// Mitsubishi GX Works2 project: SmartFarmDXST   PLC: FX3U/FX3UC

// global labels: Global1
VAR_GLOBAL
  v1 enb AT M130 : BOOL;
  v1 mode slc AT M131 : BOOL;
  v1 man OD AT M132 : BOOL;
  v1 Temp1 AT M133 : BOOL;
  v1 Temp2 AT M134 : BOOL;
  v1 Humid1 AT M135 : BOOL;
  v1 Humid2 AT M136 : BOOL;
  v1 Time1 AT M137 : BOOL;
  v1 Time2 AT M138 : BOOL;
  v1 Time3 AT M139 : BOOL;
  v1 Time4 AT M140 : BOOL;
  v1 AMB config AT M141 : BOOL;
  v1 TIME config AT M142 : BOOL;
  v1 con pass flg AT M144 : BOOL;
  v1 Drv flg AT M145 : BOOL;
  v1 Yman OD AT M146 : BOOL;
  v1 run dur AT D102 : INT;
  v1 rest dur AT D103 : INT;
  v0 enb AT M100 : BOOL;
  v0 mode slc AT M101 : BOOL;
  v0 man OD AT M102 : BOOL;
  v0 Temp1 AT M103 : BOOL;
  v0 Temp2 AT M104 : BOOL;
  v0 Humid1 AT M105 : BOOL;
  v0 Humid2 AT M106 : BOOL;
  v0 Time1 AT M107 : BOOL;
  v0 Time2 AT M108 : BOOL;
  v0 Time3 AT M109 : BOOL;
  v0 Time4 AT M110 : BOOL;
  v0 AMB config AT M111 : BOOL;
  v0 TIME config AT M112 : BOOL;
  v0 con kill flg AT M113 : BOOL;
  v0 con pass flg AT M114 : BOOL;
  v0 Drv flg AT M115 : BOOL;
  v0 run dur AT D100 : INT;
  v0 rest dur AT D101 : INT;
  v0 Yman OD AT M116 : BOOL;
  v1 con kill flg AT M143 : BOOL;
  AmbSens1 Humid AT D10 : INT;
  AmbSens1 Temp AT D11 : INT;
  AmbSens2 Humid AT D12 : INT;
  AmbSens2 Temp AT D13 : INT;
  SoilSens1 moist AT D20 : INT;
  SoilSens1 temp AT D21 : INT;
  SoilSens1 cond AT D22 : INT;
  SoilSens1 PH AT D23 : INT;
  SoilSens1 N AT D24 : INT;
  SoilSens1 P AT D25 : INT;
  SoilSens1 K AT D26 : INT;
  TempCon1 minT AT D30 : INT;
  TempCon1 maxT AT D31 : INT;
  TempCon1 Flg AT M10 : BOOL;
  TempCon1 Hs AT D32 : INT;
  TempCon1 Ms AT D33 : INT;
  TempCon1 Ss AT D34 : INT;
  TempCon1 He AT D35 : INT;
  TempCon1 Me AT D36 : INT;
  TempCon1 Se AT D37 : INT;
  TempCon2 minT AT D38 : INT;
  TempCon2 maxT AT D39 : INT;
  TempCon2 Flg AT M20 : BOOL;
  TempCon2 Hs AT D40 : INT;
  TempCon2 Ms AT D41 : INT;
  TempCon2 Ss AT D42 : INT;
  TempCon2 He AT D43 : INT;
  TempCon2 Me AT D44 : INT;
  TempCon2 Se AT D45 : INT;
  HumidCon1 minH AT D46 : INT;
  HumidCon1 maxH AT D47 : INT;
  HumidCon1 Flg AT M30 : BOOL;
  HumidCon1 Hs AT D48 : INT;
  HumidCon1 Ms AT D49 : INT;
  HumidCon1 Ss AT D50 : INT;
  HumidCon1 He AT D51 : INT;
  HumidCon1 Me AT D52 : INT;
  HumidCon1 Se AT D53 : INT;
  HumidCon2 minH AT D54 : INT;
  HumidCon2 maxH AT D55 : INT;
  HumidCon2 Flg AT M40 : BOOL;
  HumidCon2 Hs AT D56 : INT;
  HumidCon2 Ms AT D57 : INT;
  HumidCon2 Ss AT D58 : INT;
  HumidCon2 He AT D59 : INT;
  HumidCon2 Me AT D60 : INT;
  HumidCon2 Se AT D61 : INT;
  TimeCon1 Flg AT M50 : BOOL;
  TimeCon1 Hs AT D62 : INT;
  TimeCon1 Ms AT D63 : INT;
  TimeCon1 Ss AT D64 : INT;
  TimeCon2 Flg AT M60 : BOOL;
  TimeCon2 Hs AT D68 : INT;
  TimeCon2 Ms AT D69 : INT;
  TimeCon2 Ss AT D70 : INT;
  TimeCon3 Flg AT M70 : BOOL;
  TimeCon3 Hs AT D74 : INT;
  TimeCon3 Ms AT D75 : INT;
  TimeCon3 Ss AT D76 : INT;
  TimeCon4 Flg AT M80 : BOOL;
  TimeCon4 Hs AT D80 : INT;
  TimeCon4 Ms AT D81 : INT;
  TimeCon4 Ss AT D82 : INT;
  TimeCon1 He AT D65 : INT;
  TimeCon1 Me AT D66 : INT;
  TimeCon1 Se AT D67 : INT;
END_VAR
VAR (*class 0*)
  TimeCon2 He AT D71 : INT;
  TimeCon2 Me AT D72 : INT;
  TimeCon2 Se AT D73 : INT;
  TimeCon3 He AT D77 : INT;
  TimeCon3 Me AT D78 : INT;
END_VAR
VAR_GLOBAL
  TimeCon3 Se AT D79 : INT;
END_VAR
VAR (*class 0*)
  TimeCon4 He AT D83 : INT;
  TimeCon4 Me AT D84 : INT;
END_VAR
VAR_GLOBAL
  TimeCon4 Se AT D85 : INT;
END_VAR

// task Task_01 (event TRUE, interval 0, priority 31): Valve0

PROGRAM Valve0
(* structured ladder/FBD written out as ST: instructions are called as NAME(EN, inputs, outputs); _pN, _eN, _tN stand for wires *)
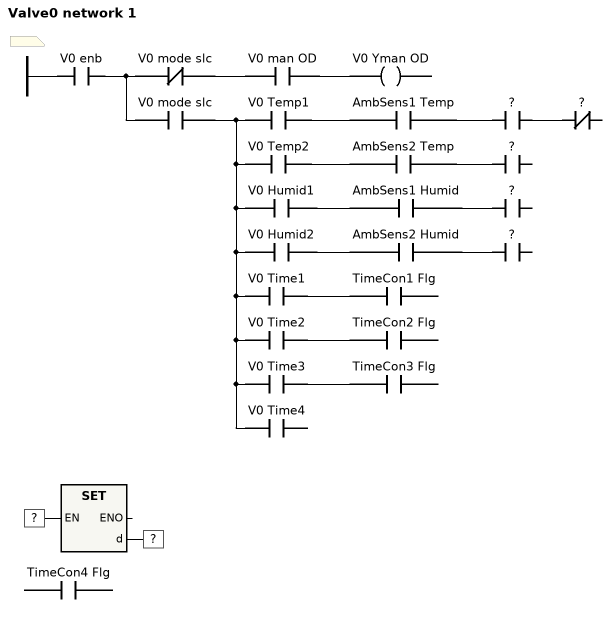
(* network 1 *)
(*  *)
_p1 := V0 enb;
V0 Yman OD := _p1 AND NOT V0 mode slc AND V0 man OD;
SET(?, ?);
(* not connected to any output: V0 mode slc, V0 Temp1, AmbSens1 Temp, ?, ?, V0 Temp2, AmbSens2 Temp, ?, V0 Humid1, AmbSens1 Humid, ?, V0 Humid2, AmbSens2 Humid, ?, V0 Time1, TimeCon1 Flg, V0 Time2, TimeCon2 Flg, V0 Time3, TimeCon3 Flg, V0 Time4, TimeCon4 Flg *)
END_PROGRAM
